{attribute 'Tc2GvlVarNames'}
VAR_CONFIG
END_VAR

(* stored: Version 1.1.0.1, ProductVersion 3.1.4024.15
   GVL Variable_Configuration: Id {c9e841e3-1c97-41bd-b566-916d88a97c8a} *)
